FUNCTION_BLOCK CAT1 (* Composite Function Block Type *)
  (* Standard: 61499-2 *)
  (* Version 0.0, 10/08/2022, Pranay Jhunjhunwala, Schneider Electric, template *)
  PACKAGE Main;
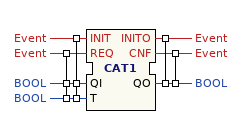
  EVENT_INPUT
    INIT WITH QI, T; (* Initialization Request *)
    REQ WITH QI, T; (* Normal Execution Request *)
  END_EVENT
  EVENT_OUTPUT
    INITO WITH QO; (* Initialization Confirm *)
    CNF WITH QO; (* Execution Confirmation *)
  END_EVENT
  VAR_INPUT
    QI : BOOL; (* Input event qualifier *)
    T : BOOL;
  END_VAR
  VAR_OUTPUT
    QO : BOOL; (* Output event qualifier *)
  END_VAR
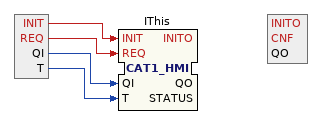
  FBS
    IThis : CAT1_HMI;
  END_FBS
  EVENT_CONNECTIONS
    INIT TO IThis.INIT;
    REQ TO IThis.REQ;
  END_CONNECTIONS
  DATA_CONNECTIONS
    QI TO IThis.QI;
    T TO IThis.T;
  END_CONNECTIONS
END_FUNCTION_BLOCK
